Fanuc KAREL source: kt00906.KL

-- PROVISIONAL review KL for V940-1; original PC SHA256 b9a11ff28ef6aea9adc8f33a265fd39d6714429592b12586568240f077c6d887
-- Incomplete behavior may be omitted. Consult companion uncertainty JSON. Do not deploy.
PROGRAM KT00906
%NOLOCKGROUP
BEGIN
  -- V9_ZERO_TABLE_METADATA_HINT layout=0002_ascii; no indexed target words; source/name/runtime held
  -- UNRESOLVED_PC offsets 5-31; opcodes 27,27,49,7E,AD,31,4A
  -- UNRESOLVED_PC offsets 36-40; opcodes 7F
END KT00906
